Staubli VAL3: delete.pgx

public program delete(string x_sName, num x_nResult)
  local string l_sItem
  local num l_nDefault
begin
  //
  // delete the select program in
  //
  if isDefined(saveProg:pProg[x_sName])
    // delete
    delete(saveProg:pProg[x_sName])
  endIf
end
